FUNCTION_BLOCK VALVE_VIEW (* Valve Position Display *)
  (* Standard: 61499-1 *)
  (* Version 0.2, 2010-12-12, JHC, Holobloc Inc, Removed INIT WITH POS - position not updated. *)
  (* Version 0.1, 2004-09-01, JHC, Rockwell Automation, Deleted QI,QO; initialized DIA:=0.. *)
  (* Version 0.0, 2000-05-01, JHC, Rockwell Automation *)
  (* Compiler header: package fb.rt.process; *)
  (* Compiler Java Sun JDK 1.6.0 *)
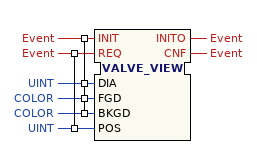
  EVENT_INPUT
    INIT WITH DIA, FGD, BKGD; (* Initialization *)
    REQ WITH POS; (* Request *)
  END_EVENT
  EVENT_OUTPUT
    INITO; (* Initialization Confirm *)
    CNF; (* Service Confirmation *)
  END_EVENT
  VAR_INPUT
    DIA : UINT; (* View height/width in pixels *)
    FGD : COLOR := COLOR#blue; (* Shaft body color *)
    BKGD : COLOR := COLOR#white; (* Background color *)
    POS : UINT; (* Current valve position *)
  END_VAR
END_FUNCTION_BLOCK
